// TwinCAT 3 PLC project Untitled1
// ProgramVersion: 3.1.4026.14
// libraries:
//   Tc2_Standard, * (Beckhoff Automation GmbH)
//   Tc2_System, * (Beckhoff Automation GmbH)
//   Tc3_Database, * (Beckhoff Automation GmbH)
//   Tc3_EventLogger, * (Beckhoff Automation GmbH)
// project tree:
//   DUTs/ DUT_SQL.TcDUT (not stored)
//   / PlcTask.TcTTO (not stored)
//   POUs/ MAIN.TcPOU, FC_SQL_InsertCommands.TcPOU

// ---- POUs/MAIN.TcPOU
PROGRAM MAIN
VAR
    FB_SQLDatabaseEvt : FB_SQLDatabaseEvt(sNetID := '', tTimeout := T#5S);
    FB_SQLCommandEvt  : FB_SQLCommandEvt(sNetID := '', tTimeout := T#5S);
    FB_SQLResultEvt   : FB_SQLResultEvt(sNetID := '', tTimeout := T#5S);

    iStep: INT;
    SQL_Commands: ARRAY[1..2] OF STRING(255);
    iSampleNr: INT := 1;
    iSensorValue: INT := 5431;
    sSelectDataCommand : STRING(255);
END_VAR


CASE iStep OF
    0:
        iStep := 10;

    10: // Connect to Database
        FB_SQLDatabaseEvt.Connect(hDBID := 1);
        IF FB_SQLDatabaseEvt.bConnected THEN
            iStep := 20;
        END_IF

    20: // Create SQL Command Object
        FB_SQLDatabaseEvt.CreateCmd(pSQLCommand := ADR(FB_SQLCommandEvt));
        IF NOT FB_SQLDatabaseEvt.bBusy THEN
            iStep := 30;
        END_IF

    30: // Generate INSERT Commands
        SQL_Commands[1] := FC_SQL_InsertCommands(iSensorValue, iSampleNr);
        iStep := 40;

    40: // Execute Insert Command
        IF FB_SQLCommandEvt.Execute(pSQLCmd := ADR(SQL_Commands[1]), cbSQLCmd := SIZEOF(SQL_Commands[1])) THEN
            iStep := 50;
        END_IF

    50: // Prepare SELECT Query
        sSelectDataCommand := 'SELECT TOP 10 * FROM [db_accessadmin].[TempSensor_Data] ORDER BY Time DESC;';
        iStep := 60;

    60: // Execute SELECT Command
         FB_SQLCommandEvt.ExecuteDataReturn(
            pSQLCmd := ADR(sSelectDataCommand),
            cbSQLCmd := SIZEOF(sSelectDataCommand),
            pSQLDBResult := ADR(FB_SQLResultEvt)); 
        
   

END_CASE

END_PROGRAM

// ---- POUs/FC_SQL_InsertCommands.TcPOU
FUNCTION FC_SQL_InsertCommands : STRING(255)
VAR_INPUT
    iSensorValue: INT;
    iSampleNr: INT;
END_VAR

FC_SQL_InsertCommands := 'INSERT INTO [db_accessadmin].[TempSensor_Data] (SensorValue, SampleNr, Time) VALUES (';
FC_SQL_InsertCommands := CONCAT(FC_SQL_InsertCommands, INT_TO_STRING(iSensorValue));
FC_SQL_InsertCommands := CONCAT(FC_SQL_InsertCommands, ', ');
FC_SQL_InsertCommands := CONCAT(FC_SQL_InsertCommands, INT_TO_STRING(iSampleNr));
FC_SQL_InsertCommands := CONCAT(FC_SQL_InsertCommands, ', GETDATE());');

END_FUNCTION
